// TIA Portal V16 export
// export: Created 2024-12-03T15:41:46.6092365Z, ExportSetting WithReadOnly, DisplayName Totally Integrated Automation Portal, DisplayVersion V16 Update 6, DisplayName TIA Portal Version Control Interface, DisplayVersion V16 Update 2, DisplayName TIA Portal Openness, DisplayVersion V16 Update 6, DisplayName TIA Portal Teamcenter Gateway, DisplayVersion V16, DisplayName SINAMICS Startdrive Advanced, DisplayVersion V16 Update 5, DisplayName SINAMICS Startdrive G130, G150, S120, S150, SINAMICS MV, S210, DisplayVersion V16 Update 5, DisplayName SINAMICS Startdrive G110M, G120, G120C, G120D, G120P, G115D, DisplayVersion V16 Update 5, DisplayName STEP 7 Professional, DisplayVersion V16 Update 6, DisplayName STEP 7 Safety, DisplayVersion V16, DisplayName WinCC Advanced / Unified PC, DisplayVersion V16 Update 6
VAR_GLOBAL   // PLC tag table "01 MainRack"
   I_EMG_MAIN AT %I7124.0 : Bool;
   I_EMG_ZONE_5B AT %I7124.5 : Bool;
   I_EMG_ZONE_3_4 AT %I7124.1 : Bool;
   I_EMG_ZONE_5 AT %I7124.4 : Bool;
   I_EMG_ZONE_2B AT %I7124.3 : Bool;
   I_EMG_ZONE_2A AT %I7124.2 : Bool;
   Q_RESET_EMG AT %Q6946.0 : Bool;
   Q_LED_GREEN AT %Q6946.2 : Bool;
   Q_LED_ORANGE AT %Q6946.3 : Bool;
   Q_LED_RED AT %Q6946.1 : Bool;
END_VAR
